// SIMATIC S7-200 project (STEP 7-Micro/WIN), CPU 224 REL 02.01

SYMBOL_TABLE USER1
tempUp           I0.1     // Zwieksz temperarture docelowa
tempDown         I0.2     // Zmniejsz temperature docelowa
histUp           I0.3     // zwieksz histereze
histDown         I0.4     // zmniejsz histereze
odczytTemp       AIW8     // odczyt z pt 100
grzalka          Q0.2     // uruchomienie grzalki
flaga_wiatrak    V0.0
flaga_grzalka    V0.1
flaga_idle       V0.2
IDLE             Q0.3     // stan bezczynnosci
set_IDLE         M0.1
reset_IDLE       M0.2
set_grza³ka      M0.3
reset_grza³ka    M0.4
set_wentylator   M0.5
reset_wentylator M0.6
wentylator       Q0.1     // uruchomienie wentylatora
END_SYMBOL_TABLE

ORGANIZATION_BLOCK MAIN:OB1
TITLE=PROGRAM COMMENTS
BEGIN
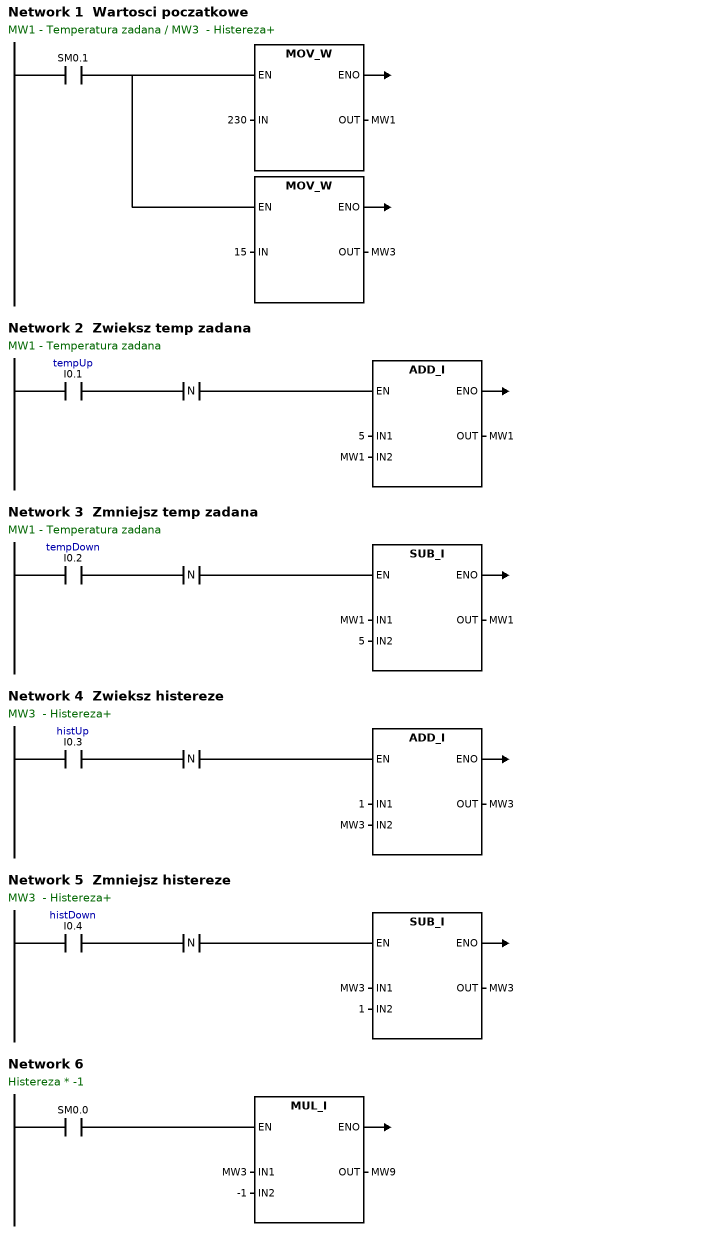
Network 1 // Wartosci poczatkowe
// MW1 - Temperatura zadana
// MW3  - Histereza+
LD     SM0.1
MOVW   230, MW1
MOVW   15, MW3
Network 2 // Zwieksz temp zadana
// MW1 - Temperatura zadana
LD     tempUp:I0.1
ED
+I     5, MW1
Network 3 // Zmniejsz temp zadana
// MW1 - Temperatura zadana
LD     tempDown:I0.2
ED
-I     5, MW1
Network 4 // Zwieksz histereze
// MW3  - Histereza+
LD     histUp:I0.3
ED
+I     1, MW3
Network 5 // Zmniejsz histereze
// MW3  - Histereza+
LD     histDown:I0.4
ED
-I     1, MW3
Network 6
// Histereza * -1
LD     SM0.0
MOVW   MW3, MW9
*I     -1, MW9
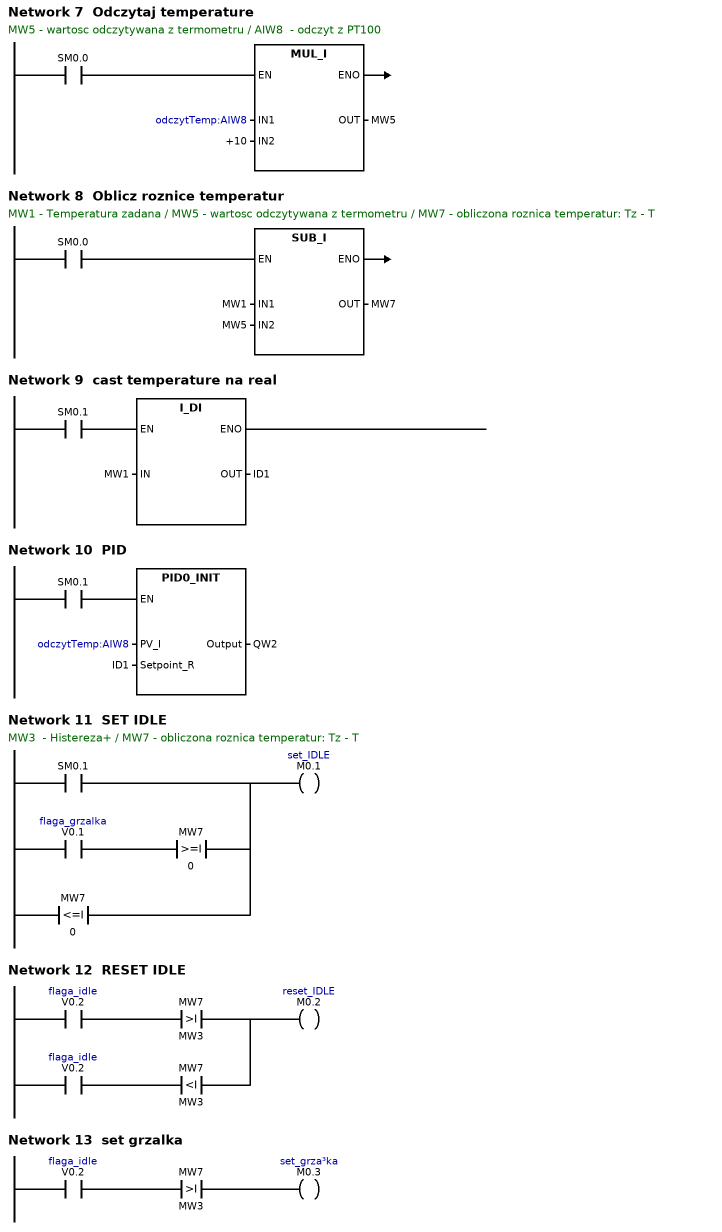
Network 7 // Odczytaj temperature
// MW5 - wartosc odczytywana z termometru
// AIW8  - odczyt z PT100
LD     SM0.0
MOVW   odczytTemp:AIW8, MW5
*I     +10, MW5
Network 8 // Oblicz roznice temperatur
// MW1 - Temperatura zadana
// MW5 - wartosc odczytywana z termometru
// MW7 - obliczona roznica temperatur: Tz - T
LD     SM0.0
MOVW   MW1, MW7
-I     MW5, MW7
Network 9 // cast temperature na real
// (network saved uncompiled; LAD cells follow)
// row 0: c0 -| |- SM0.1  c1 [I_DI EN:=power@row0, IN:=MW1, ENO=>power, OUT=>ID1]  c2 --  c3 --
// row 1: c1 [box]
Network 10 // PID
// (network saved uncompiled; LAD cells follow)
// row 0: c0 -| |- SM0.1  c1 [PID0_INIT EN:=power@row0, PV_I:=odczytTemp:AIW8, Setpoint_R:=ID1, Output=>QW2]
// row 1: c1 [box]
Network 11 // SET IDLE
// MW3  - Histereza+
// MW7 - obliczona roznica temperatur: Tz - T
LD     SM0.1
LD     flaga_grzalka:V0.1
AW>=   MW7, 0
OLD
OW<=   MW7, 0
=      set_IDLE:M0.1
Network 12 // RESET IDLE
LD     flaga_idle:V0.2
AW>    MW7, MW3
LD     flaga_idle:V0.2
AW<    MW7, MW3
OLD
=      reset_IDLE:M0.2
Network 13 // set grzalka
LD     flaga_idle:V0.2
AW>    MW7, MW3
=      set_grza³ka:M0.3
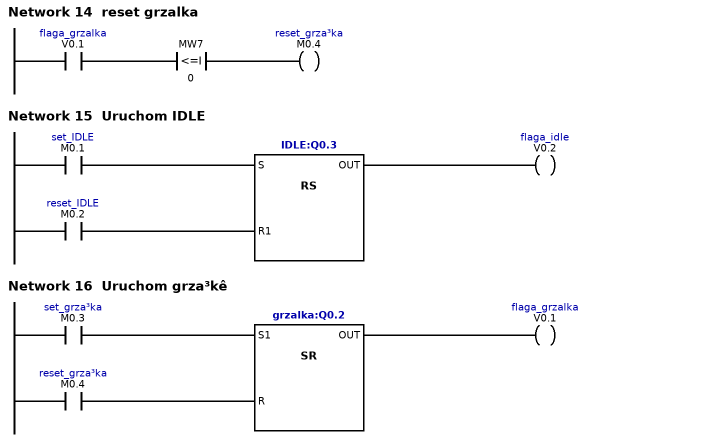
Network 14 // reset grzalka
LD     flaga_grzalka:V0.1
AW<=   MW7, 0
=      reset_grza³ka:M0.4
Network 15 // Uruchom IDLE
LD     set_IDLE:M0.1
LD     reset_IDLE:M0.2
NOT
LPS
A      IDLE:Q0.3
=      IDLE:Q0.3
LPP
ALD
O      IDLE:Q0.3
=      IDLE:Q0.3
=      flaga_idle:V0.2
Network 16 // Uruchom grza³kê
LD     set_grza³ka:M0.3
LD     reset_grza³ka:M0.4
NOT
A      grzalka:Q0.2
OLD
=      grzalka:Q0.2
=      flaga_grzalka:V0.1
END_ORGANIZATION_BLOCK

// SBR1: protected block, not included

// INT1: protected block, not included

// (further data pages could not be read)
